TYPE ModbusReal :
UNION
	rawdata		: ARRAY[0..1] OF WORD;
	value		: REAL;
END_UNION
END_TYPE

(* stored: Version 1.1.0.1
   DUT ModbusReal: Id {593612c3-a13d-4bbd-a6bb-d8e9bb5c86f3} *)
